FUNCTION_BLOCK PuestoManualV2
VAR_INPUT
	SFCreset:BOOL;
	Reset:BOOL;
	Enable:BOOL;
	FinCiclo:BOOL;
	SensorPallet:BOOL;
	Pulsador1 AT %I*:BOOL;
	ModoDoble:BOOL;
	NumeroDePuesto :INT;
	
END_VAR
VAR_OUTPUT
	StopperOFF AT %Q*:BOOL;
	Centrador AT%Q*:BOOL;
	LuzRoja AT%Q*:BOOL;
	FinPuesto:BOOL;
	SalidaAlarma:BOOL;
	EnMovimiento:BOOL;
	EsperandoPalet :BOOL;
END_VAR
VAR
END_VAR

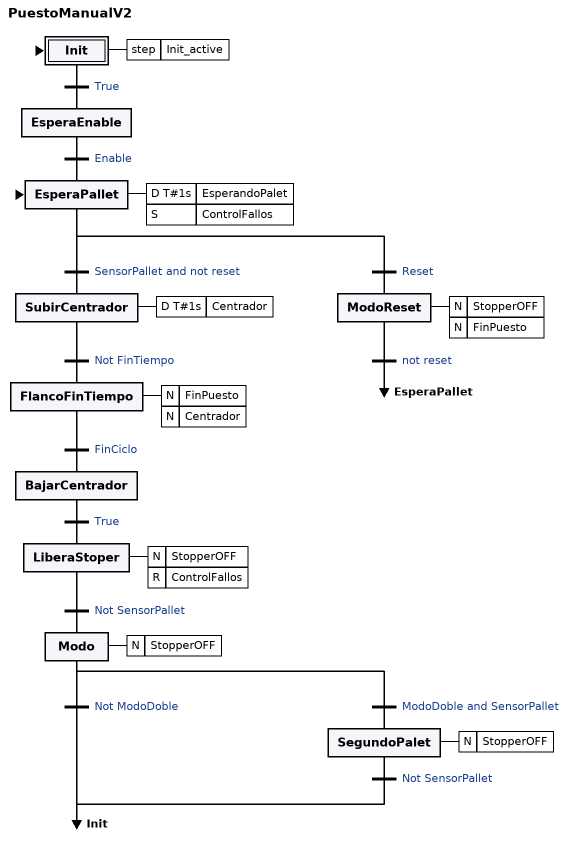
INITIAL_STEP Init:
    Init_active(N);  // step action
END_STEP
TRANSITION FROM Init TO EsperaEnable
    := True;
END_TRANSITION
STEP EsperaEnable:
END_STEP
TRANSITION FROM EsperaEnable TO EsperaPallet
    := Enable;
END_TRANSITION
STEP EsperaPallet:
    EsperandoPalet(D, T#1s);
    ControlFallos(S);
END_STEP
TRANSITION FROM EsperaPallet TO SubirCentrador
    := SensorPallet and not reset;
END_TRANSITION
STEP SubirCentrador:  // min time T#1s
    Centrador(D, T#1s);
END_STEP
TRANSITION FROM SubirCentrador TO FlancoFinTiempo
    := Not FinTiempo;
END_TRANSITION
STEP FlancoFinTiempo:
    FinPuesto(N);
    Centrador(N);
END_STEP
TRANSITION FROM FlancoFinTiempo TO BajarCentrador
    := FinCiclo;
END_TRANSITION
STEP BajarCentrador:  // min time T#1s
END_STEP
TRANSITION FROM BajarCentrador TO LiberaStoper
    := True;
END_TRANSITION
TRANSITION FROM EsperaPallet TO ModoReset
    := Reset;
END_TRANSITION
STEP ModoReset:
    StopperOFF(N);
    FinPuesto(N);
END_STEP
TRANSITION FROM ModoReset TO EsperaPallet
    := not reset;
END_TRANSITION
STEP LiberaStoper:  // min time T#1s
    StopperOFF(N);
    ControlFallos(R);
END_STEP
TRANSITION FROM LiberaStoper TO Modo
    := Not SensorPallet;
END_TRANSITION
STEP Modo:
    StopperOFF(N);
END_STEP
TRANSITION FROM Modo TO Init
    := Not ModoDoble;
END_TRANSITION
TRANSITION FROM Modo TO SegundoPalet
    := ModoDoble and SensorPallet;
END_TRANSITION
STEP SegundoPalet:  // min time T#1s
    StopperOFF(N);
END_STEP
TRANSITION FROM SegundoPalet TO Init
    := Not SensorPallet;
END_TRANSITION

ACTION ControlFallos:

IF GVL.FalloPallet[NumeroDePuesto] THEN
	LuzRoja :=TRUE;
	FinPuesto := FALSE;
ELSE
	LuzRoja :=TRUE;
	FinPuesto := FALSE;
END_IF


IF GVL.FalloPallet[NumeroDePuesto] AND Pulsador1 THEN
	GVL.FalloPallet[NumeroDePuesto] := FALSE;
END_IF
END_ACTION

ACTION Init_active:
LuzRoja := FALSE;
FinPUesto :=FALSE;
SFCreset:=FALSE;
END_ACTION

END_FUNCTION_BLOCK

(* stored: Version 1.1.0.1, ProductVersion 3.1.4024.3
   POU PuestoManualV2: Id {6f175889-191b-40e7-86e0-b25d8d32ac31}, SpecialFunc None
   Action ControlFallos: Id {ead04932-3073-49e8-8935-cae11b4e9846}
   Action Init_active: Id {a6553785-f09e-4c60-afcf-db7cbd880a72} *)
